// TIA Portal V20 export
// export: Created 2026-04-18T06:34:09.8141714Z, ExportSetting WithDefaults, DisplayName Totally Integrated Automation Portal, DisplayVersion V20, DisplayName TIA Portal Openness, DisplayVersion V20, DisplayName TIA Portal Version Control Interface, DisplayVersion V20, DisplayName STEP 7 Professional, DisplayVersion V20, DisplayName STEP 7 Safety, DisplayVersion V20, DisplayName WinCC Basic/Comfort/Advanced, DisplayVersion V20
DATA_BLOCK "DB_ProcessPlant_A1"   // DB4
{ S7_Optimized_Access := 'TRUE' }
VERSION : 0.1
// stored: AutoNumber true, DBAccessibleFromOPCUA true, DBAccessibleFromWebserver true, IsOnlyStoredInLoadMemory false, IsRetainMemResEnabled false, IsWriteProtectedInAS false, MemoryReserve 100
   VAR
      plantId : Int := 1;
      plantName : String[32] := 'Plant A1';
      units { S7_SetPoint := 'True'} : Array[1..2] of "UDT_ProcessUnit";
   END_VAR
BEGIN
   units[1].unitId := 1;
   units[2].unitId := 2;
   units[1].unitName := 'Reactor R-100';
   units[2].unitName := 'Reactor R-200';
   units[1].recipeId := 101;
   units[2].recipeId := 201;
   units[1].modules[1].moduleId := 11;
   units[1].modules[2].moduleId := 12;
   units[1].modules[3].moduleId := 13;
   units[2].modules[1].moduleId := 21;
   units[2].modules[2].moduleId := 22;
   units[2].modules[3].moduleId := 23;
   units[1].modules[1].moduleName := 'Dosing Station DS-01';
   units[1].modules[2].moduleName := 'Heating Module HM-01';
   units[1].modules[3].moduleName := 'Agitator AG-01';
   units[2].modules[1].moduleName := 'Dosing Station DS-02';
   units[2].modules[2].moduleName := 'Heating Module HM-02';
   units[2].modules[3].moduleName := 'Agitator AG-02';
   units[1].modules[1].moduleType := 1;
   units[1].modules[2].moduleType := 2;
   units[1].modules[3].moduleType := 3;
   units[2].modules[1].moduleType := 1;
   units[2].modules[2].moduleType := 2;
   units[2].modules[3].moduleType := 3;
   units[1].modules[1].valves[1].valveTag := 'V-10101';
   units[1].modules[1].valves[2].valveTag := 'V-10102';
   units[1].modules[1].valves[3].valveTag := 'V-10103';
   units[1].modules[1].valves[4].valveTag := 'V-10104';
   units[1].modules[2].valves[1].valveTag := 'V-10201';
   units[1].modules[2].valves[2].valveTag := 'V-10202';
   units[1].modules[2].valves[3].valveTag := 'V-10203';
   units[1].modules[2].valves[4].valveTag := 'V-10204';
   units[1].modules[3].valves[1].valveTag := 'V-10301';
   units[1].modules[3].valves[2].valveTag := 'V-10302';
   units[1].modules[3].valves[3].valveTag := 'V-10303';
   units[1].modules[3].valves[4].valveTag := 'V-10304';
   units[2].modules[1].valves[1].valveTag := 'V-20101';
   units[2].modules[1].valves[2].valveTag := 'V-20102';
   units[2].modules[1].valves[3].valveTag := 'V-20103';
   units[2].modules[1].valves[4].valveTag := 'V-20104';
   units[2].modules[2].valves[1].valveTag := 'V-20201';
   units[2].modules[2].valves[2].valveTag := 'V-20202';
   units[2].modules[2].valves[3].valveTag := 'V-20203';
   units[2].modules[2].valves[4].valveTag := 'V-20204';
   units[2].modules[3].valves[1].valveTag := 'V-20301';
   units[2].modules[3].valves[2].valveTag := 'V-20302';
   units[2].modules[3].valves[3].valveTag := 'V-20303';
   units[2].modules[3].valves[4].valveTag := 'V-20304';
   units[1].modules[1].valves[1..2].valveType := 4;
   units[1].modules[1].valves[3..4].valveType := 1;
   units[1].modules[2].valves[1..2].valveType := 2;
   units[1].modules[2].valves[3..4].valveType := 1;
   units[1].modules[3].valves[1..4].valveType := 3;
   units[2].modules[1].valves[1..2].valveType := 4;
   units[2].modules[1].valves[3..4].valveType := 1;
   units[2].modules[2].valves[1..2].valveType := 2;
   units[2].modules[2].valves[3..4].valveType := 1;
   units[2].modules[3].valves[1..4].valveType := 3;
END_DATA_BLOCK
